{attribute 'qualified_only'}
{attribute 'strict'}
TYPE E_FunctionForkOrder :
(
	E_ORDER_UNKNOWN,
	E_ORDER_CENTER,
	E_ORDER_LEFT,
	E_ORDER_RIGHT
);
END_TYPE

(* stored: Version 1.1.0.1, ProductVersion 3.1.4024.9
   DUT E_FunctionForkOrder: Id {1f01a1e1-8a68-416a-9f8b-b8ae133cb6a0} *)
